Yaskawa INFORM job: VIK.JBI

/JOB
//NAME VIK
//POS
///NPOS 14,14,14,3,0,0
///TOOL 0
///POSTYPE PULSE
///PULSE
C00000=-44188,-83847,-61893,31337,114325,-33875
C00001=-43194,-84730,-62262,31667,113761,-33613
C00002=-44187,-83848,-61893,31338,114326,-33873
C00003=-44187,-83095,-60119,31153,113720,-34057
C00004=-44188,-83847,-61893,31337,114325,-33875
C00005=-38294,-69301,-55326,34501,114941,-31029
C00006=-37385,-70057,-55693,34765,114435,-30789
C00007=-38295,-69303,-55327,34501,114941,-31029
C00008=-38295,-68744,-53650,34283,114322,-31243
C00009=-38295,-69303,-55327,34501,114941,-31029
C00010=-46527,-81632,-60952,30529,115665,-34498
C00011=-44038,-85471,-61764,31141,113480,-34070
C00012=-37221,-68411,-54090,34763,114250,-30783
C00013=-39345,-63825,-52880,34517,116453,-30987
BC00000=353550,856982,323391
BC00001=353550,856982,323391
BC00002=353550,856982,323389
BC00003=353550,856982,323389
BC00004=353550,856982,323391
BC00005=353550,856982,323391
BC00006=353550,856982,323391
BC00007=353550,856982,323391
BC00008=353550,856982,323391
BC00009=353550,856982,323391
BC00010=353550,856982,323388
BC00011=353550,856982,323388
BC00012=353550,856982,323388
BC00013=353550,856982,323388
EC00000=1,1
EC00001=1,1
EC00002=2,1
EC00003=2,1
EC00004=1,1
EC00005=1,1
EC00006=1,1
EC00007=1,1
EC00008=1,1
EC00009=1,1
EC00010=1,1
EC00011=1,1
EC00012=1,1
EC00013=1,1
///POSTYPE BASE
///RECTAN
///RCONF 0,0,0,0,0,0,0,0,0,0,0,0,0,0,0,0,0,0,0,0,0,0,0,0
P00006=0.222,-3.123,-1.508,0.0000,0.0000,0.0000
P00051=0.367,3.892,0.009,0.0000,0.0000,0.0000
P00052=0.088,2.832,-0.342,0.0000,0.0000,0.0000
//INST
///DATE 2024/05/16 12:02
///ATTR SC,RW
///GROUP1 RB1,BS1
///GROUP2 ST1
NOP
CALL JOB:CLEAN-R1_KM_NEW
SFTOF3D
SMOVL C00000 BC00000 V=100.0  +MOVJ EC00000
SREFP 3 C00001 BC00001  +REFP EC00001
CALL JOB:SEARCH-R1-S13D_TEST
SET P051 P006
SFTON3D P051
SMOVL C00002 BC00002 V=100.0  +MOVJ EC00002
SREFP 3 C00003 BC00003  +REFP EC00003
CALL JOB:SEARCH-R1-S13D_TEST
SET P051 P006
SFTON3D P051
SMOVL C00004 BC00004 V=100.0  +MOVJ EC00004
SFTOF3D
SMOVL C00005 BC00005 V=100.0  +MOVJ EC00005
SREFP 3 C00006 BC00006  +REFP EC00006
CALL JOB:SEARCH-R1-S13D_TEST
SET P052 P006
SFTON3D P052
SMOVL C00007 BC00007 V=100.0  +MOVJ EC00007
SREFP 3 C00008 BC00008  +REFP EC00008
CALL JOB:SEARCH-R1-S13D_TEST
SET P052 P006
SFTON3D P052
SFTOF3D
SMOVL C00009 BC00009 V=100.0  +MOVJ EC00009
SMOVL C00010 BC00010 V=166.7  +MOVJ EC00010
SFTON3D P051
SMOVL C00011 BC00011 V=166.7  +MOVJ EC00011
SFTON3D P052
SMOVL C00012 BC00012 V=8.3  +MOVJ EC00012
SFTOF3D
SMOVL C00013 BC00013 V=166.7  +MOVJ EC00013
END
